(* CoDeSys 2.3.9.62 project: 0750-0881.WagoAppKNX.SunshadeActuator.pro *)
(* Libraries: C:\Work\WAGO\WAGO.Sandbox\WAGO.KNX\CoDeSys\2.3\mod_com.lib, C:\Work\WAGO\WAGO.Sandbox\WAGO.KNX\CoDeSys\2.3\KNX_Standard.lib 27.4.23 16:22:16, WAGOLibKNXDevice.lib 23.1.08 13:40:44, SysLibGetAddress.lib 7.9.10 15:37:47, C:\Work\WAGO\WAGO.Sandbox\WAGO.KNX\CoDeSys\2.3\KNX_Applikations_02.lib 27.4.23 16:22:16, C:\Work\WAGO\WAGO.Sandbox\WAGO.KNX\CoDeSys\2.3\DALI_02.lib 27.4.23 16:22:16, Standard.lib, SYSLIBCALLBACK.LIB *)

(* PLC configuration (modules and I/O channels)
0753-0646 KNX-TP1 [Type_30_1_Channels] node 1, in %IB0 out %QB0 {INTTypePAAssignment = PLC; INTTypeModule = plugged}
  AT %IB0 [BYTEOnB_I] First Byte of 24
  AT %QB0 [BYTEOnB_Q] First Byte of 24
Fieldbus variables [FB_VARS] node 1, in %IB0 out %QB0
Flag variables [FLAG_VARS] node 2, in %IB0 out %QB0
Modbus-Master [MB_MASTER] node 3, in %IB0 out %QB0
*)

(* POU PLC_PRG, ST *)
PROGRAM PLC_PRG
VAR
END_VAR
KNX1_Master_646(
	bModule_753_646:=1,
	typKNX:=typKNX1,
	enumStatusKNX=>enumStatusKNX1,
	xProg_Mode=>xProg_ModeKNX1);
END_PROGRAM

(* POU PLC_PRG_CFC, CFC *)
PROGRAM PLC_PRG_CFC
VAR
END_VAR
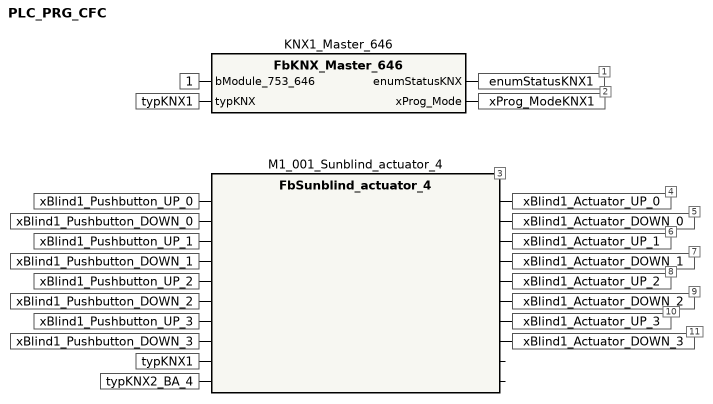
_CFC_ (* Continuous Function Chart, elements in execution order *)
#0 KNX1_Master_646:FbKNX_Master_646(bModule_753_646: 1, typKNX: typKNX1)
#1 enumStatusKNX1 <= #0.enumStatusKNX
#2 xProg_ModeKNX1 <= #0.xProg_Mode
#3 M1_001_Sunblind_actuator_4:FbSunblind_actuator_4(xBlind1_Pushbutton_UP_0, xBlind1_Pushbutton_DOWN_0, xBlind1_Pushbutton_UP_1, xBlind1_Pushbutton_DOWN_1, xBlind1_Pushbutton_UP_2, xBlind1_Pushbutton_DOWN_2, xBlind1_Pushbutton_UP_3, xBlind1_Pushbutton_DOWN_3, typKNX1, typKNX2_BA_4)
#4 xBlind1_Actuator_UP_0 <= #3.out 1
#5 xBlind1_Actuator_DOWN_0 <= #3.out 2
#6 xBlind1_Actuator_UP_1 <= #3.out 3
#7 xBlind1_Actuator_DOWN_1 <= #3.out 4
#8 xBlind1_Actuator_UP_2 <= #3.out 5
#9 xBlind1_Actuator_DOWN_2 <= #3.out 6
#10 xBlind1_Actuator_UP_3 <= #3.out 7
#11 xBlind1_Actuator_DOWN_3 <= #3.out 8
_END_CFC_
END_PROGRAM
